// TIA Portal V18 export
FUNCTION_BLOCK "SireneMain"   // FB6, FBD
{ S7_Optimized_Access := 'TRUE' }
VERSION : 0.1
// stored: AutoNumber true, IsIECCheckEnabled false, IsRetainMemResEnabled false, MemoryReserve 100, SetENOAutomatically false, UDAEnableTagReadback false
   VAR
      sirene_Instance { S7_SetPoint := 'True'} : "sirene_v2";
   END_VAR
BEGIN

REGION Network 2: Trigger
END_REGION

REGION Network 3
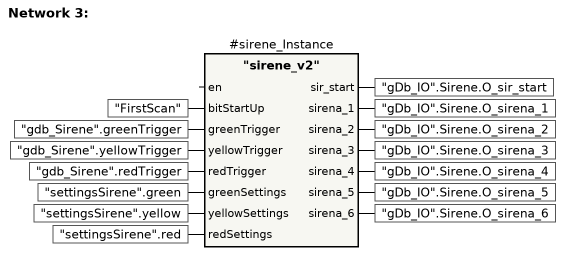
   #sirene_Instance(bitStartUp := "FirstScan",   // "sirene_v2"
                    greenTrigger := "gdb_Sirene".greenTrigger,
                    yellowTrigger := "gdb_Sirene".yellowTrigger,
                    redTrigger := "gdb_Sirene".redTrigger,
                    greenSettings := "settingsSirene".green,
                    yellowSettings := "settingsSirene".yellow,
                    redSettings := "settingsSirene".red,
                    sir_start => "gDb_IO".Sirene.O_sir_start,
                    sirena_1 => "gDb_IO".Sirene.O_sirena_1,
                    sirena_2 => "gDb_IO".Sirene.O_sirena_2,
                    sirena_3 => "gDb_IO".Sirene.O_sirena_3,
                    sirena_4 => "gDb_IO".Sirene.O_sirena_4,
                    sirena_5 => "gDb_IO".Sirene.O_sirena_5,
                    sirena_6 => "gDb_IO".Sirene.O_sirena_6);
END_REGION
END_FUNCTION_BLOCK
